(* IEC 61131-3 sources: CodesysTest/export/Function Blocks/IO/FB_PhysicalDigitalInput.pou/IsOff.prop, 1 file *)

(* ---- Get.pm.st ---- *)
(*#-#-#-#-#-#-#-#-#-#---Declaration---#-#-#-#-#-#-#-#-#-#-#-#-#*)

VAR
END_VAR
(*#-#-#-#-#-#-#-#-#-#---Implementation---#-#-#-#-#-#-#-#-#-#-#-#-#*)

IsOff := NOT Active;
